TYPE DUT_SQL :
STRUCT
    SensorValue : INT;
    SampleNr : INT;
    Timestamp : STRING(50);
END_STRUCT
END_TYPE

(* stored: Version 1.1.0.1
   DUT DUT_SQL: Id {388cf1ad-db44-4458-b218-2f70112d1464} *)
